Yaskawa INFORM job: linear_start.JBI

/JOB
//NAME AAA
//POS
///NPOS 1,0,0,0,0,0
C00000=-50237,120156,80713,3485,-54801,-4055
//INST
///DATE 2023/02/07 09:04
///ATTR SC,RW
///GROUP1 RB1
NOP
MOVJ C00000 VJ=1.0 PL=0
END
